// TIA Portal V18 export
// export: Created 2026-06-23T08:49:31.0010641Z, ExportSetting WithDefaults, DisplayName Totally Integrated Automation Portal, DisplayVersion V18, DisplayName TIA Portal Openness, DisplayVersion V18, DisplayName TIA Portal Version Control Interface, DisplayVersion V18, DisplayName STEP 7 Professional, DisplayVersion V18, DisplayName STEP 7 Safety, DisplayVersion V18, DisplayName WinCC Professional, DisplayVersion V18
ORGANIZATION_BLOCK "OB30_PID_PLC1_Bon2"   // OB30, LAD, CyclicInterrupt
{ S7_Optimized_Access := 'TRUE' }
VERSION : 0.1
// stored: AutoNumber true, IsIECCheckEnabled false, SetENOAutomatically false
   VAR_INPUT
      Initial_Call : Bool;   // Initial call of this OB
      Event_Count : Int;   // Events discarded
   END_VAR
BEGIN

REGION Network 1: Initialize PID Bon 2 Kp parameter
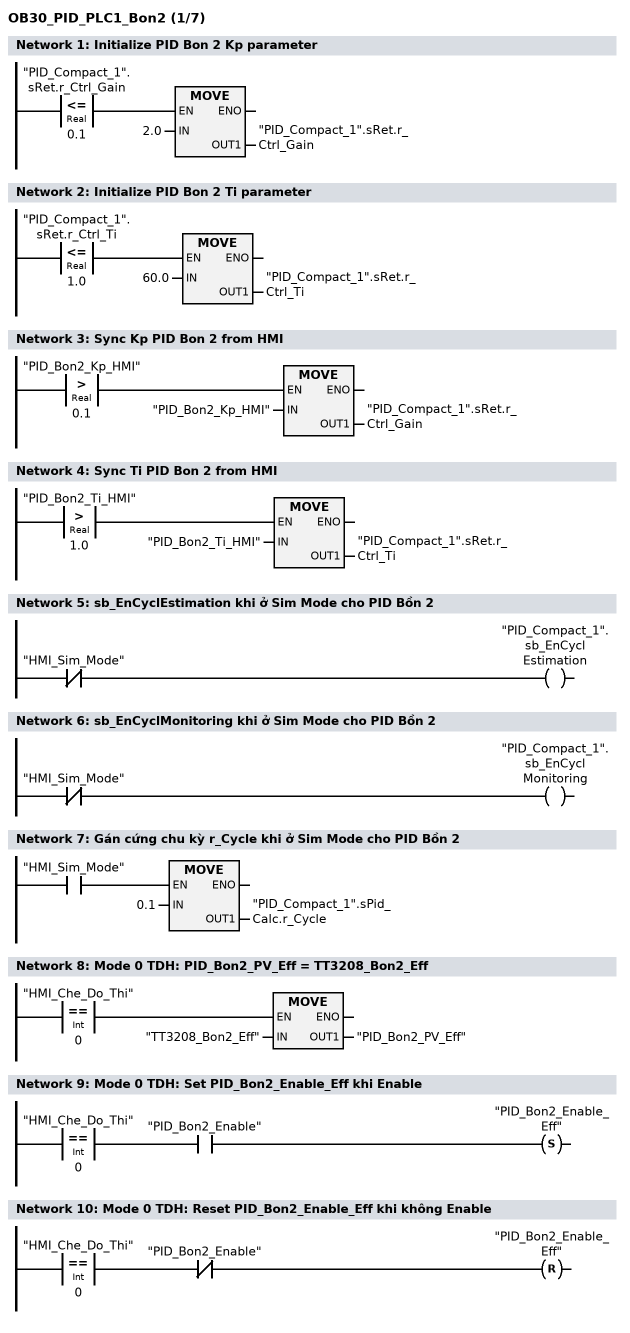
   RUNG wire#powerrail
      { S7_Templates := "SrcType := Real" } LE_Contact(in1 := "PID_Compact_1".sRet.r_Ctrl_Gain, in2 := 0.1)
      { S7_GenerateENO := "TRUE" } Move(in := 2.0, out1 => "PID_Compact_1".sRet.r_Ctrl_Gain)
   END_RUNG
   // the same network as SCL:
   IF "PID_Compact_1".sRet.r_Ctrl_Gain <= 0.1 THEN "PID_Compact_1".sRet.r_Ctrl_Gain := 2.0; END_IF;
END_REGION

REGION Network 2: Initialize PID Bon 2 Ti parameter
   RUNG wire#powerrail
      { S7_Templates := "SrcType := Real" } LE_Contact(in1 := "PID_Compact_1".sRet.r_Ctrl_Ti, in2 := 1.0)
      { S7_GenerateENO := "TRUE" } Move(in := 60.0, out1 => "PID_Compact_1".sRet.r_Ctrl_Ti)
   END_RUNG
   // the same network as SCL:
   IF "PID_Compact_1".sRet.r_Ctrl_Ti <= 1.0 THEN "PID_Compact_1".sRet.r_Ctrl_Ti := 60.0; END_IF;
END_REGION

REGION Network 3: Sync Kp PID Bon 2 from HMI
   RUNG wire#powerrail
      { S7_Templates := "SrcType := Real" } GT_Contact(in1 := "PID_Bon2_Kp_HMI", in2 := 0.1)
      { S7_GenerateENO := "TRUE" } Move(in := "PID_Bon2_Kp_HMI", out1 => "PID_Compact_1".sRet.r_Ctrl_Gain)
   END_RUNG
   // the same network as SCL:
   IF "PID_Bon2_Kp_HMI" > 0.1 THEN "PID_Compact_1".sRet.r_Ctrl_Gain := "PID_Bon2_Kp_HMI"; END_IF;
END_REGION

REGION Network 4: Sync Ti PID Bon 2 from HMI
   RUNG wire#powerrail
      { S7_Templates := "SrcType := Real" } GT_Contact(in1 := "PID_Bon2_Ti_HMI", in2 := 1.0)
      { S7_GenerateENO := "TRUE" } Move(in := "PID_Bon2_Ti_HMI", out1 => "PID_Compact_1".sRet.r_Ctrl_Ti)
   END_RUNG
   // the same network as SCL:
   IF "PID_Bon2_Ti_HMI" > 1.0 THEN "PID_Compact_1".sRet.r_Ctrl_Ti := "PID_Bon2_Ti_HMI"; END_IF;
END_REGION

REGION Network 5: sb_EnCyclEstimation khi ở Sim Mode cho PID Bồn 2
   RUNG wire#powerrail
      I_Contact( "HMI_Sim_Mode" )
      Coil( "PID_Compact_1".sb_EnCyclEstimation )
   END_RUNG
   // the same network as SCL:
   "PID_Compact_1".sb_EnCyclEstimation := NOT "HMI_Sim_Mode";
END_REGION

REGION Network 6: sb_EnCyclMonitoring khi ở Sim Mode cho PID Bồn 2
   RUNG wire#powerrail
      I_Contact( "HMI_Sim_Mode" )
      Coil( "PID_Compact_1".sb_EnCyclMonitoring )
   END_RUNG
   // the same network as SCL:
   "PID_Compact_1".sb_EnCyclMonitoring := NOT "HMI_Sim_Mode";
END_REGION

REGION Network 7: Gán cứng chu kỳ r_Cycle khi ở Sim Mode cho PID Bồn 2
   RUNG wire#powerrail
      Contact( "HMI_Sim_Mode" )
      { S7_GenerateENO := "TRUE" } Move(in := 0.1, out1 => "PID_Compact_1".sPid_Calc.r_Cycle)
   END_RUNG
   // the same network as SCL:
   IF "HMI_Sim_Mode" THEN "PID_Compact_1".sPid_Calc.r_Cycle := 0.1; END_IF;
END_REGION

REGION Network 8: Mode 0 TDH: PID_Bon2_PV_Eff = TT3208_Bon2_Eff
   RUNG wire#powerrail
      { S7_Templates := "SrcType := Int" } EQ_Contact(in1 := "HMI_Che_Do_Thi", in2 := 0)
      { S7_GenerateENO := "TRUE" } Move(in := "TT3208_Bon2_Eff", out1 => "PID_Bon2_PV_Eff")
   END_RUNG
   // the same network as SCL:
   IF "HMI_Che_Do_Thi" = 0 THEN "PID_Bon2_PV_Eff" := "TT3208_Bon2_Eff"; END_IF;
END_REGION

REGION Network 9: Mode 0 TDH: Set PID_Bon2_Enable_Eff khi Enable
   RUNG wire#powerrail
      { S7_Templates := "SrcType := Int" } EQ_Contact(in1 := "HMI_Che_Do_Thi", in2 := 0)
      Contact( "PID_Bon2_Enable" )
      S_Coil( "PID_Bon2_Enable_Eff" )
   END_RUNG
   // the same network as SCL:
   IF ("HMI_Che_Do_Thi" = 0) AND "PID_Bon2_Enable" THEN "PID_Bon2_Enable_Eff" := TRUE; END_IF;
END_REGION

REGION Network 10: Mode 0 TDH: Reset PID_Bon2_Enable_Eff khi không Enable
   RUNG wire#powerrail
      { S7_Templates := "SrcType := Int" } EQ_Contact(in1 := "HMI_Che_Do_Thi", in2 := 0)
      I_Contact( "PID_Bon2_Enable" )
      R_Coil( "PID_Bon2_Enable_Eff" )
   END_RUNG
   // the same network as SCL:
   IF ("HMI_Che_Do_Thi" = 0) AND NOT "PID_Bon2_Enable" THEN "PID_Bon2_Enable_Eff" := FALSE; END_IF;
END_REGION

REGION Network 11: Mode 1 DN: PID_Bon2_PV_Eff = VFD_Bon2_Actual_Speed_Feedback
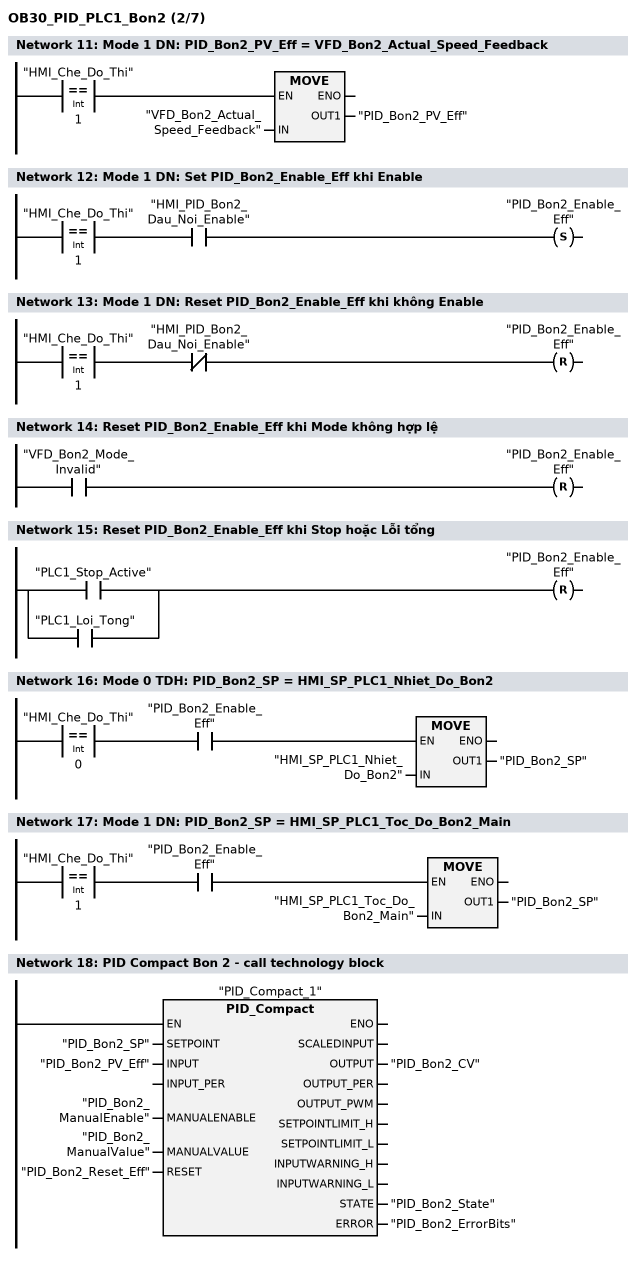
   RUNG wire#powerrail
      { S7_Templates := "SrcType := Int" } EQ_Contact(in1 := "HMI_Che_Do_Thi", in2 := 1)
      { S7_GenerateENO := "TRUE" } Move(in := "VFD_Bon2_Actual_Speed_Feedback", out1 => "PID_Bon2_PV_Eff")
   END_RUNG
   // the same network as SCL:
   IF "HMI_Che_Do_Thi" = 1 THEN "PID_Bon2_PV_Eff" := "VFD_Bon2_Actual_Speed_Feedback"; END_IF;
END_REGION

REGION Network 12: Mode 1 DN: Set PID_Bon2_Enable_Eff khi Enable
   RUNG wire#powerrail
      { S7_Templates := "SrcType := Int" } EQ_Contact(in1 := "HMI_Che_Do_Thi", in2 := 1)
      Contact( "HMI_PID_Bon2_Dau_Noi_Enable" )
      S_Coil( "PID_Bon2_Enable_Eff" )
   END_RUNG
   // the same network as SCL:
   IF ("HMI_Che_Do_Thi" = 1) AND "HMI_PID_Bon2_Dau_Noi_Enable" THEN "PID_Bon2_Enable_Eff" := TRUE; END_IF;
END_REGION

REGION Network 13: Mode 1 DN: Reset PID_Bon2_Enable_Eff khi không Enable
   RUNG wire#powerrail
      { S7_Templates := "SrcType := Int" } EQ_Contact(in1 := "HMI_Che_Do_Thi", in2 := 1)
      I_Contact( "HMI_PID_Bon2_Dau_Noi_Enable" )
      R_Coil( "PID_Bon2_Enable_Eff" )
   END_RUNG
   // the same network as SCL:
   IF ("HMI_Che_Do_Thi" = 1) AND NOT "HMI_PID_Bon2_Dau_Noi_Enable" THEN
       "PID_Bon2_Enable_Eff" := FALSE;
   END_IF;
END_REGION

REGION Network 14: Reset PID_Bon2_Enable_Eff khi Mode không hợp lệ
   RUNG wire#powerrail
      Contact( "VFD_Bon2_Mode_Invalid" )
      R_Coil( "PID_Bon2_Enable_Eff" )
   END_RUNG
   // the same network as SCL:
   IF "VFD_Bon2_Mode_Invalid" THEN "PID_Bon2_Enable_Eff" := FALSE; END_IF;
END_REGION

REGION Network 15: Reset PID_Bon2_Enable_Eff khi Stop hoặc Lỗi tổng
   RUNG wire#powerrail
      Contact( "PLC1_Stop_Active" )
      wire#w1
      R_Coil( "PID_Bon2_Enable_Eff" )
   END_RUNG
   RUNG wire#powerrail
      Contact( "PLC1_Loi_Tong" )
   END_RUNG wire#w1
   // the same network as SCL:
   IF "PLC1_Stop_Active" OR "PLC1_Loi_Tong" THEN "PID_Bon2_Enable_Eff" := FALSE; END_IF;
END_REGION

REGION Network 16: Mode 0 TDH: PID_Bon2_SP = HMI_SP_PLC1_Nhiet_Do_Bon2
   RUNG wire#powerrail
      { S7_Templates := "SrcType := Int" } EQ_Contact(in1 := "HMI_Che_Do_Thi", in2 := 0)
      Contact( "PID_Bon2_Enable_Eff" )
      { S7_GenerateENO := "TRUE" } Move(in := "HMI_SP_PLC1_Nhiet_Do_Bon2", out1 => "PID_Bon2_SP")
   END_RUNG
   // the same network as SCL:
   IF ("HMI_Che_Do_Thi" = 0) AND "PID_Bon2_Enable_Eff" THEN
       "PID_Bon2_SP" := "HMI_SP_PLC1_Nhiet_Do_Bon2";
   END_IF;
END_REGION

REGION Network 17: Mode 1 DN: PID_Bon2_SP = HMI_SP_PLC1_Toc_Do_Bon2_Main
   RUNG wire#powerrail
      { S7_Templates := "SrcType := Int" } EQ_Contact(in1 := "HMI_Che_Do_Thi", in2 := 1)
      Contact( "PID_Bon2_Enable_Eff" )
      { S7_GenerateENO := "TRUE" } Move(in := "HMI_SP_PLC1_Toc_Do_Bon2_Main", out1 => "PID_Bon2_SP")
   END_RUNG
   // the same network as SCL:
   IF ("HMI_Che_Do_Thi" = 1) AND "PID_Bon2_Enable_Eff" THEN
       "PID_Bon2_SP" := "HMI_SP_PLC1_Toc_Do_Bon2_Main";
   END_IF;
END_REGION

REGION Network 18: PID Compact Bon 2 - call technology block
   RUNG wire#powerrail
      "PID_Compact_1".PID_Compact(Setpoint := "PID_Bon2_SP", Input := "PID_Bon2_PV_Eff", Input_PER :=, ManualEnable := "PID_Bon2_ManualEnable", ManualValue := "PID_Bon2_ManualValue", Reset := "PID_Bon2_Reset_Eff", ScaledInput =>, Output => "PID_Bon2_CV", Output_PER =>, Output_PWM =>, SetpointLimit_H =>, SetpointLimit_L =>, InputWarning_H =>, InputWarning_L =>, State => "PID_Bon2_State", Error => "PID_Bon2_ErrorBits")
   END_RUNG
   // the same network as SCL:
   "PID_Compact_1"(Setpoint := "PID_Bon2_SP",   // PID_Compact
                   Input := "PID_Bon2_PV_Eff",
                   ManualEnable := "PID_Bon2_ManualEnable",
                   ManualValue := "PID_Bon2_ManualValue",
                   Reset := "PID_Bon2_Reset_Eff",
                   Output => "PID_Bon2_CV",
                   State => "PID_Bon2_State",
                   Error => "PID_Bon2_ErrorBits");
END_REGION

REGION Network 19: Detect PID Bon 2 Error
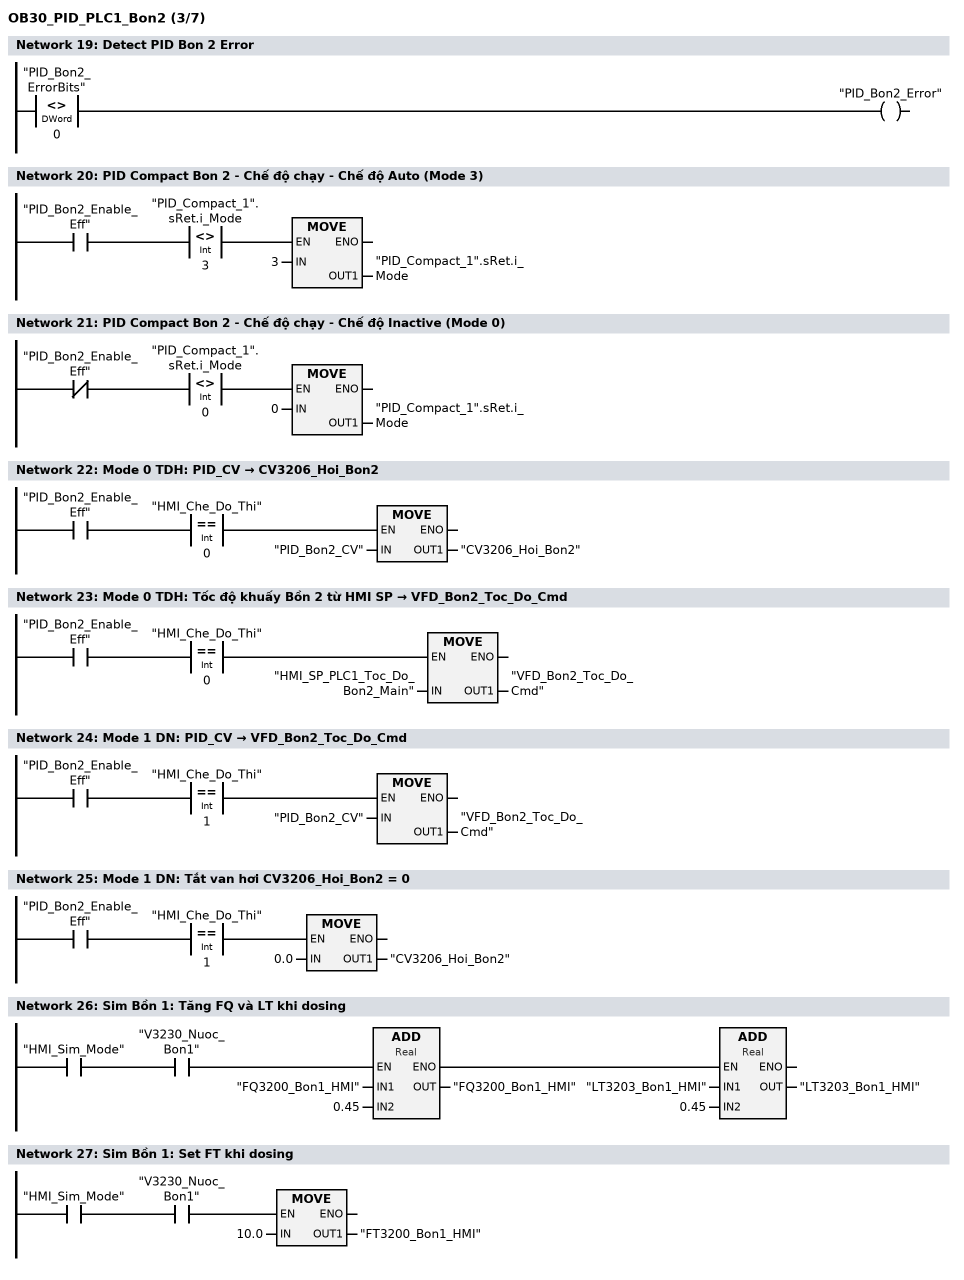
   RUNG wire#powerrail
      { S7_Templates := "SrcType := DWord" } NE_Contact(in1 := "PID_Bon2_ErrorBits", in2 := 0)
      Coil( "PID_Bon2_Error" )
   END_RUNG
   // the same network as SCL:
   "PID_Bon2_Error" := "PID_Bon2_ErrorBits" <> 0;
END_REGION

REGION Network 20: PID Compact Bon 2 - Chế độ chạy - Chế độ Auto (Mode 3)
   RUNG wire#powerrail
      Contact( "PID_Bon2_Enable_Eff" )
      { S7_Templates := "SrcType := Int" } NE_Contact(in1 := "PID_Compact_1".sRet.i_Mode, in2 := 3)
      { S7_GenerateENO := "TRUE" } Move(in := 3, out1 => "PID_Compact_1".sRet.i_Mode)
   END_RUNG
   // the same network as SCL:
   IF "PID_Bon2_Enable_Eff" AND ("PID_Compact_1".sRet.i_Mode <> 3) THEN
       "PID_Compact_1".sRet.i_Mode := 3;
   END_IF;
END_REGION

REGION Network 21: PID Compact Bon 2 - Chế độ chạy - Chế độ Inactive (Mode 0)
   RUNG wire#powerrail
      I_Contact( "PID_Bon2_Enable_Eff" )
      { S7_Templates := "SrcType := Int" } NE_Contact(in1 := "PID_Compact_1".sRet.i_Mode, in2 := 0)
      { S7_GenerateENO := "TRUE" } Move(in := 0, out1 => "PID_Compact_1".sRet.i_Mode)
   END_RUNG
   // the same network as SCL:
   IF NOT "PID_Bon2_Enable_Eff" AND ("PID_Compact_1".sRet.i_Mode <> 0) THEN
       "PID_Compact_1".sRet.i_Mode := 0;
   END_IF;
END_REGION

REGION Network 22: Mode 0 TDH: PID_CV → CV3206_Hoi_Bon2
   RUNG wire#powerrail
      Contact( "PID_Bon2_Enable_Eff" )
      { S7_Templates := "SrcType := Int" } EQ_Contact(in1 := "HMI_Che_Do_Thi", in2 := 0)
      { S7_GenerateENO := "TRUE" } Move(in := "PID_Bon2_CV", out1 => "CV3206_Hoi_Bon2")
   END_RUNG
   // the same network as SCL:
   IF "PID_Bon2_Enable_Eff" AND ("HMI_Che_Do_Thi" = 0) THEN "CV3206_Hoi_Bon2" := "PID_Bon2_CV"; END_IF;
END_REGION

REGION Network 23: Mode 0 TDH: Tốc độ khuấy Bồn 2 từ HMI SP → VFD_Bon2_Toc_Do_Cmd
   RUNG wire#powerrail
      Contact( "PID_Bon2_Enable_Eff" )
      { S7_Templates := "SrcType := Int" } EQ_Contact(in1 := "HMI_Che_Do_Thi", in2 := 0)
      { S7_GenerateENO := "TRUE" } Move(in := "HMI_SP_PLC1_Toc_Do_Bon2_Main", out1 => "VFD_Bon2_Toc_Do_Cmd")
   END_RUNG
   // the same network as SCL:
   IF "PID_Bon2_Enable_Eff" AND ("HMI_Che_Do_Thi" = 0) THEN
       "VFD_Bon2_Toc_Do_Cmd" := "HMI_SP_PLC1_Toc_Do_Bon2_Main";
   END_IF;
END_REGION

REGION Network 24: Mode 1 DN: PID_CV → VFD_Bon2_Toc_Do_Cmd
   RUNG wire#powerrail
      Contact( "PID_Bon2_Enable_Eff" )
      { S7_Templates := "SrcType := Int" } EQ_Contact(in1 := "HMI_Che_Do_Thi", in2 := 1)
      { S7_GenerateENO := "TRUE" } Move(in := "PID_Bon2_CV", out1 => "VFD_Bon2_Toc_Do_Cmd")
   END_RUNG
   // the same network as SCL:
   IF "PID_Bon2_Enable_Eff" AND ("HMI_Che_Do_Thi" = 1) THEN "VFD_Bon2_Toc_Do_Cmd" := "PID_Bon2_CV"; END_IF;
END_REGION

REGION Network 25: Mode 1 DN: Tắt van hơi CV3206_Hoi_Bon2 = 0
   RUNG wire#powerrail
      Contact( "PID_Bon2_Enable_Eff" )
      { S7_Templates := "SrcType := Int" } EQ_Contact(in1 := "HMI_Che_Do_Thi", in2 := 1)
      { S7_GenerateENO := "TRUE" } Move(in := 0.0, out1 => "CV3206_Hoi_Bon2")
   END_RUNG
   // the same network as SCL:
   IF "PID_Bon2_Enable_Eff" AND ("HMI_Che_Do_Thi" = 1) THEN "CV3206_Hoi_Bon2" := 0.0; END_IF;
END_REGION

REGION Network 26: Sim Bồn 1: Tăng FQ và LT khi dosing
   RUNG wire#powerrail
      Contact( "HMI_Sim_Mode" )
      Contact( "V3230_Nuoc_Bon1" )
      { S7_Templates := "SrcType := Real"; S7_GenerateENO := "TRUE" } Add(in1 := "FQ3200_Bon1_HMI", in2 := 0.45, out => "FQ3200_Bon1_HMI")
      { S7_Templates := "SrcType := Real"; S7_GenerateENO := "TRUE" } Add(in1 := "LT3203_Bon1_HMI", in2 := 0.45, out => "LT3203_Bon1_HMI")
   END_RUNG
   // the same network as SCL:
   // ENO of a box is taken as its EN; it also drops when the box reports an error
   IF "HMI_Sim_Mode" AND "V3230_Nuoc_Bon1" THEN
       "FQ3200_Bon1_HMI" := "FQ3200_Bon1_HMI" + 0.45;
       "LT3203_Bon1_HMI" := "LT3203_Bon1_HMI" + 0.45;
   END_IF;
END_REGION

REGION Network 27: Sim Bồn 1: Set FT khi dosing
   RUNG wire#powerrail
      Contact( "HMI_Sim_Mode" )
      Contact( "V3230_Nuoc_Bon1" )
      { S7_GenerateENO := "TRUE" } Move(in := 10.0, out1 => "FT3200_Bon1_HMI")
   END_RUNG
   // the same network as SCL:
   IF "HMI_Sim_Mode" AND "V3230_Nuoc_Bon1" THEN "FT3200_Bon1_HMI" := 10.0; END_IF;
END_REGION

REGION Network 28: Sim Bồn 1: Reset FT khi không dosing
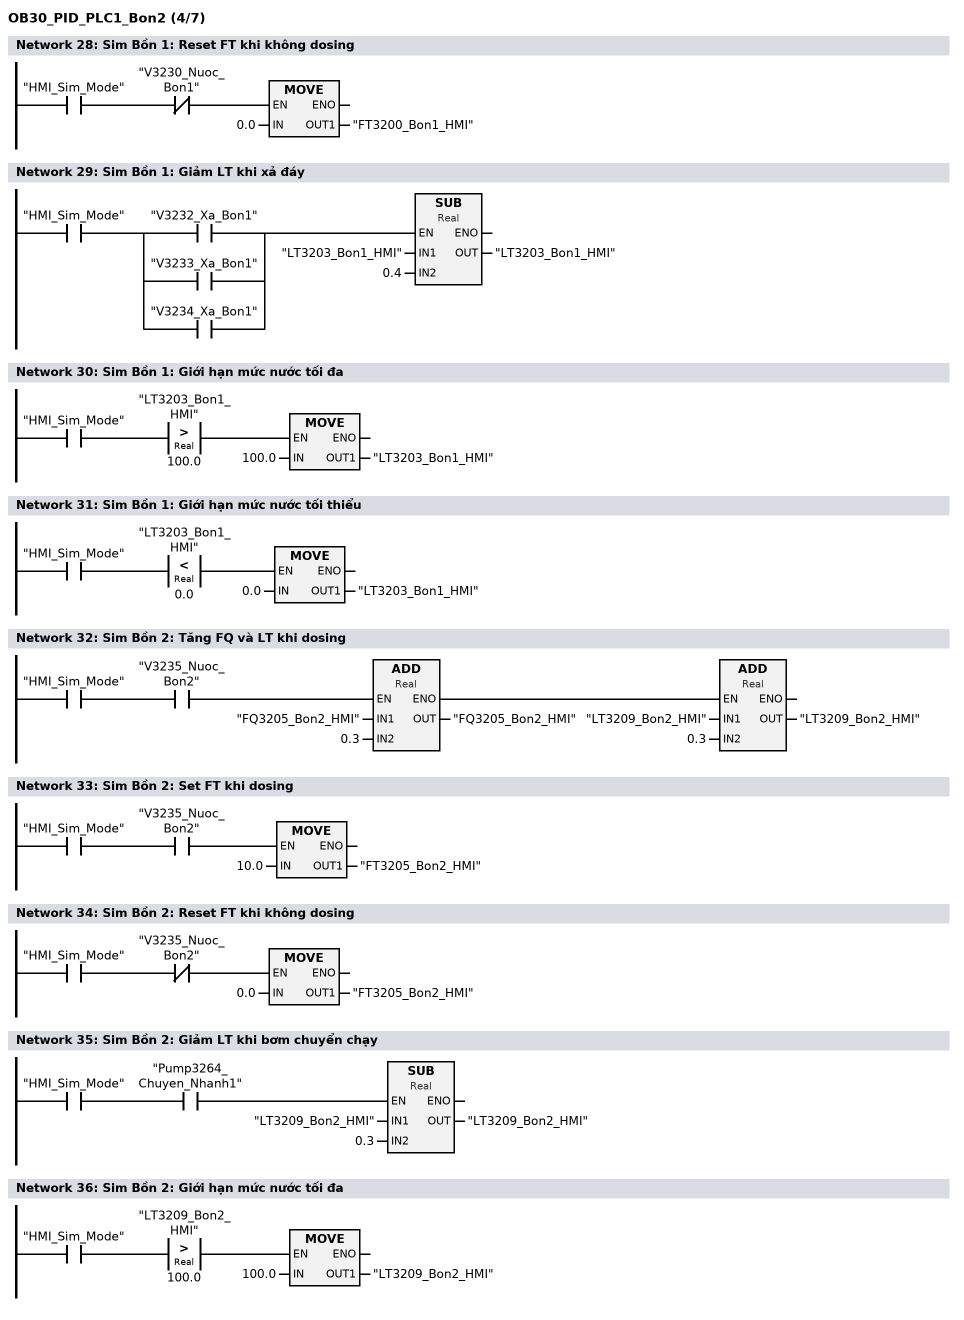
   RUNG wire#powerrail
      Contact( "HMI_Sim_Mode" )
      I_Contact( "V3230_Nuoc_Bon1" )
      { S7_GenerateENO := "TRUE" } Move(in := 0.0, out1 => "FT3200_Bon1_HMI")
   END_RUNG
   // the same network as SCL:
   IF "HMI_Sim_Mode" AND NOT "V3230_Nuoc_Bon1" THEN "FT3200_Bon1_HMI" := 0.0; END_IF;
END_REGION

REGION Network 29: Sim Bồn 1: Giảm LT khi xả đáy
   RUNG wire#powerrail
      Contact( "HMI_Sim_Mode" )
      wire#w1
      Contact( "V3232_Xa_Bon1" )
      wire#w2
      { S7_Templates := "SrcType := Real"; S7_GenerateENO := "TRUE" } Sub(in1 := "LT3203_Bon1_HMI", in2 := 0.4, out => "LT3203_Bon1_HMI")
   END_RUNG
   RUNG wire#w1
      Contact( "V3233_Xa_Bon1" )
   END_RUNG wire#w2
   RUNG wire#w1
      Contact( "V3234_Xa_Bon1" )
   END_RUNG wire#w2
   // the same network as SCL:
   IF "HMI_Sim_Mode" AND ("V3232_Xa_Bon1" OR "V3233_Xa_Bon1" OR "V3234_Xa_Bon1") THEN
       "LT3203_Bon1_HMI" := "LT3203_Bon1_HMI" - 0.4;
   END_IF;
END_REGION

REGION Network 30: Sim Bồn 1: Giới hạn mức nước tối đa
   RUNG wire#powerrail
      Contact( "HMI_Sim_Mode" )
      { S7_Templates := "SrcType := Real" } GT_Contact(in1 := "LT3203_Bon1_HMI", in2 := 100.0)
      { S7_GenerateENO := "TRUE" } Move(in := 100.0, out1 => "LT3203_Bon1_HMI")
   END_RUNG
   // the same network as SCL:
   IF "HMI_Sim_Mode" AND ("LT3203_Bon1_HMI" > 100.0) THEN "LT3203_Bon1_HMI" := 100.0; END_IF;
END_REGION

REGION Network 31: Sim Bồn 1: Giới hạn mức nước tối thiểu
   RUNG wire#powerrail
      Contact( "HMI_Sim_Mode" )
      { S7_Templates := "SrcType := Real" } LT_Contact(in1 := "LT3203_Bon1_HMI", in2 := 0.0)
      { S7_GenerateENO := "TRUE" } Move(in := 0.0, out1 => "LT3203_Bon1_HMI")
   END_RUNG
   // the same network as SCL:
   IF "HMI_Sim_Mode" AND ("LT3203_Bon1_HMI" < 0.0) THEN "LT3203_Bon1_HMI" := 0.0; END_IF;
END_REGION

REGION Network 32: Sim Bồn 2: Tăng FQ và LT khi dosing
   RUNG wire#powerrail
      Contact( "HMI_Sim_Mode" )
      Contact( "V3235_Nuoc_Bon2" )
      { S7_Templates := "SrcType := Real"; S7_GenerateENO := "TRUE" } Add(in1 := "FQ3205_Bon2_HMI", in2 := 0.3, out => "FQ3205_Bon2_HMI")
      { S7_Templates := "SrcType := Real"; S7_GenerateENO := "TRUE" } Add(in1 := "LT3209_Bon2_HMI", in2 := 0.3, out => "LT3209_Bon2_HMI")
   END_RUNG
   // the same network as SCL:
   // ENO of a box is taken as its EN; it also drops when the box reports an error
   IF "HMI_Sim_Mode" AND "V3235_Nuoc_Bon2" THEN
       "FQ3205_Bon2_HMI" := "FQ3205_Bon2_HMI" + 0.3;
       "LT3209_Bon2_HMI" := "LT3209_Bon2_HMI" + 0.3;
   END_IF;
END_REGION

REGION Network 33: Sim Bồn 2: Set FT khi dosing
   RUNG wire#powerrail
      Contact( "HMI_Sim_Mode" )
      Contact( "V3235_Nuoc_Bon2" )
      { S7_GenerateENO := "TRUE" } Move(in := 10.0, out1 => "FT3205_Bon2_HMI")
   END_RUNG
   // the same network as SCL:
   IF "HMI_Sim_Mode" AND "V3235_Nuoc_Bon2" THEN "FT3205_Bon2_HMI" := 10.0; END_IF;
END_REGION

REGION Network 34: Sim Bồn 2: Reset FT khi không dosing
   RUNG wire#powerrail
      Contact( "HMI_Sim_Mode" )
      I_Contact( "V3235_Nuoc_Bon2" )
      { S7_GenerateENO := "TRUE" } Move(in := 0.0, out1 => "FT3205_Bon2_HMI")
   END_RUNG
   // the same network as SCL:
   IF "HMI_Sim_Mode" AND NOT "V3235_Nuoc_Bon2" THEN "FT3205_Bon2_HMI" := 0.0; END_IF;
END_REGION

REGION Network 35: Sim Bồn 2: Giảm LT khi bơm chuyển chạy
   RUNG wire#powerrail
      Contact( "HMI_Sim_Mode" )
      Contact( "Pump3264_Chuyen_Nhanh1" )
      { S7_Templates := "SrcType := Real"; S7_GenerateENO := "TRUE" } Sub(in1 := "LT3209_Bon2_HMI", in2 := 0.3, out => "LT3209_Bon2_HMI")
   END_RUNG
   // the same network as SCL:
   IF "HMI_Sim_Mode" AND "Pump3264_Chuyen_Nhanh1" THEN "LT3209_Bon2_HMI" := "LT3209_Bon2_HMI" - 0.3; END_IF;
END_REGION

REGION Network 36: Sim Bồn 2: Giới hạn mức nước tối đa
   RUNG wire#powerrail
      Contact( "HMI_Sim_Mode" )
      { S7_Templates := "SrcType := Real" } GT_Contact(in1 := "LT3209_Bon2_HMI", in2 := 100.0)
      { S7_GenerateENO := "TRUE" } Move(in := 100.0, out1 => "LT3209_Bon2_HMI")
   END_RUNG
   // the same network as SCL:
   IF "HMI_Sim_Mode" AND ("LT3209_Bon2_HMI" > 100.0) THEN "LT3209_Bon2_HMI" := 100.0; END_IF;
END_REGION

REGION Network 37: Sim Bồn 2: Giới hạn mức nước tối thiểu
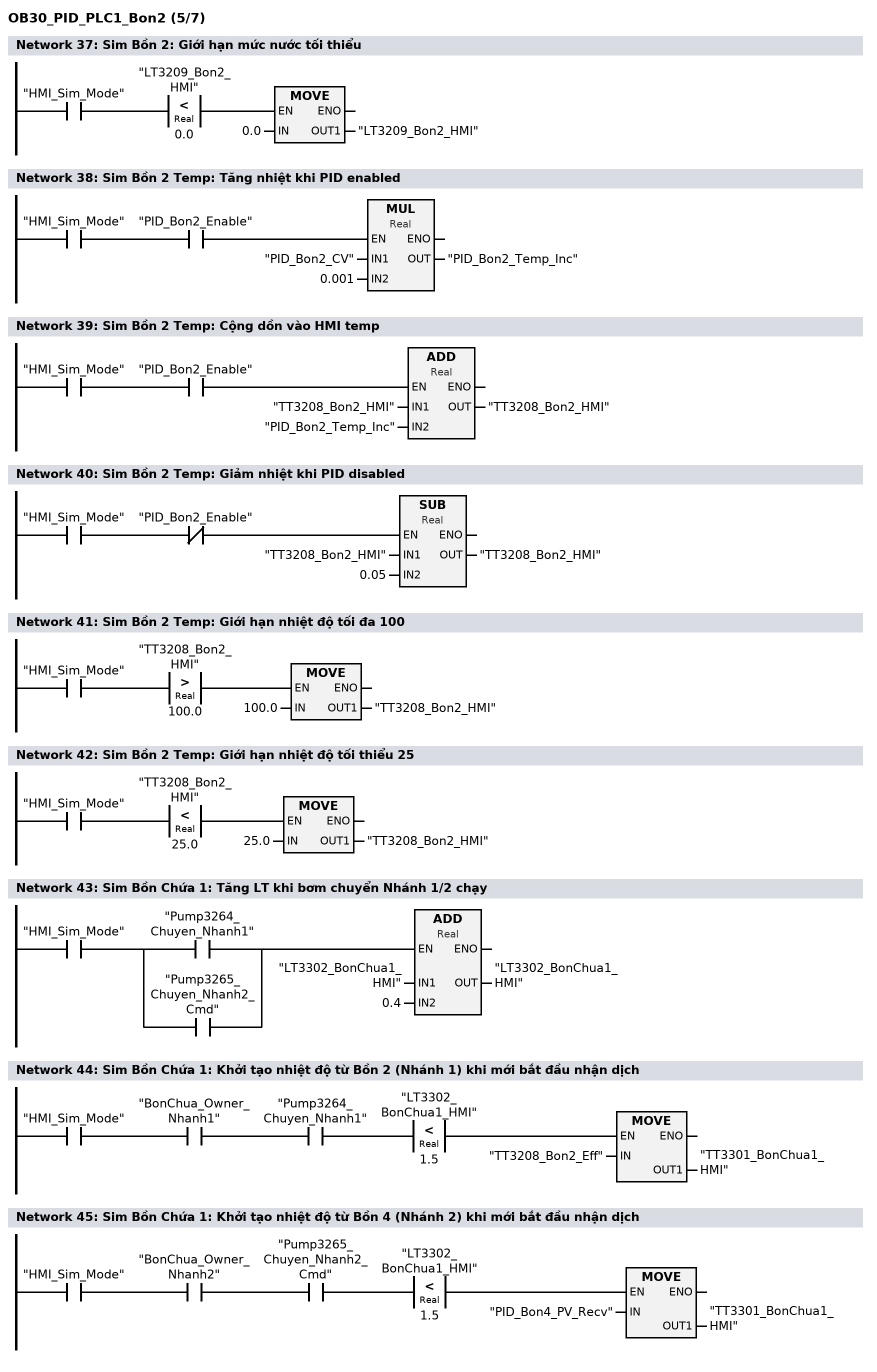
   RUNG wire#powerrail
      Contact( "HMI_Sim_Mode" )
      { S7_Templates := "SrcType := Real" } LT_Contact(in1 := "LT3209_Bon2_HMI", in2 := 0.0)
      { S7_GenerateENO := "TRUE" } Move(in := 0.0, out1 => "LT3209_Bon2_HMI")
   END_RUNG
   // the same network as SCL:
   IF "HMI_Sim_Mode" AND ("LT3209_Bon2_HMI" < 0.0) THEN "LT3209_Bon2_HMI" := 0.0; END_IF;
END_REGION

REGION Network 38: Sim Bồn 2 Temp: Tăng nhiệt khi PID enabled
   RUNG wire#powerrail
      Contact( "HMI_Sim_Mode" )
      Contact( "PID_Bon2_Enable" )
      { S7_Templates := "SrcType := Real"; S7_GenerateENO := "TRUE" } Mul(in1 := "PID_Bon2_CV", in2 := 0.001, out => "PID_Bon2_Temp_Inc")
   END_RUNG
   // the same network as SCL:
   IF "HMI_Sim_Mode" AND "PID_Bon2_Enable" THEN "PID_Bon2_Temp_Inc" := "PID_Bon2_CV" * 0.001; END_IF;
END_REGION

REGION Network 39: Sim Bồn 2 Temp: Cộng dồn vào HMI temp
   RUNG wire#powerrail
      Contact( "HMI_Sim_Mode" )
      Contact( "PID_Bon2_Enable" )
      { S7_Templates := "SrcType := Real"; S7_GenerateENO := "TRUE" } Add(in1 := "TT3208_Bon2_HMI", in2 := "PID_Bon2_Temp_Inc", out => "TT3208_Bon2_HMI")
   END_RUNG
   // the same network as SCL:
   IF "HMI_Sim_Mode" AND "PID_Bon2_Enable" THEN
       "TT3208_Bon2_HMI" := "TT3208_Bon2_HMI" + "PID_Bon2_Temp_Inc";
   END_IF;
END_REGION

REGION Network 40: Sim Bồn 2 Temp: Giảm nhiệt khi PID disabled
   RUNG wire#powerrail
      Contact( "HMI_Sim_Mode" )
      I_Contact( "PID_Bon2_Enable" )
      { S7_Templates := "SrcType := Real"; S7_GenerateENO := "TRUE" } Sub(in1 := "TT3208_Bon2_HMI", in2 := 0.05, out => "TT3208_Bon2_HMI")
   END_RUNG
   // the same network as SCL:
   IF "HMI_Sim_Mode" AND NOT "PID_Bon2_Enable" THEN "TT3208_Bon2_HMI" := "TT3208_Bon2_HMI" - 0.05; END_IF;
END_REGION

REGION Network 41: Sim Bồn 2 Temp: Giới hạn nhiệt độ tối đa 100
   RUNG wire#powerrail
      Contact( "HMI_Sim_Mode" )
      { S7_Templates := "SrcType := Real" } GT_Contact(in1 := "TT3208_Bon2_HMI", in2 := 100.0)
      { S7_GenerateENO := "TRUE" } Move(in := 100.0, out1 => "TT3208_Bon2_HMI")
   END_RUNG
   // the same network as SCL:
   IF "HMI_Sim_Mode" AND ("TT3208_Bon2_HMI" > 100.0) THEN "TT3208_Bon2_HMI" := 100.0; END_IF;
END_REGION

REGION Network 42: Sim Bồn 2 Temp: Giới hạn nhiệt độ tối thiểu 25
   RUNG wire#powerrail
      Contact( "HMI_Sim_Mode" )
      { S7_Templates := "SrcType := Real" } LT_Contact(in1 := "TT3208_Bon2_HMI", in2 := 25.0)
      { S7_GenerateENO := "TRUE" } Move(in := 25.0, out1 => "TT3208_Bon2_HMI")
   END_RUNG
   // the same network as SCL:
   IF "HMI_Sim_Mode" AND ("TT3208_Bon2_HMI" < 25.0) THEN "TT3208_Bon2_HMI" := 25.0; END_IF;
END_REGION

REGION Network 43: Sim Bồn Chứa 1: Tăng LT khi bơm chuyển Nhánh 1/2 chạy
   RUNG wire#powerrail
      Contact( "HMI_Sim_Mode" )
      wire#w1
      Contact( "Pump3264_Chuyen_Nhanh1" )
      wire#w2
      { S7_Templates := "SrcType := Real"; S7_GenerateENO := "TRUE" } Add(in1 := "LT3302_BonChua1_HMI", in2 := 0.4, out => "LT3302_BonChua1_HMI")
   END_RUNG
   RUNG wire#w1
      Contact( "Pump3265_Chuyen_Nhanh2_Cmd" )
   END_RUNG wire#w2
   // the same network as SCL:
   IF "HMI_Sim_Mode" AND ("Pump3264_Chuyen_Nhanh1" OR "Pump3265_Chuyen_Nhanh2_Cmd") THEN
       "LT3302_BonChua1_HMI" := "LT3302_BonChua1_HMI" + 0.4;
   END_IF;
END_REGION

REGION Network 44: Sim Bồn Chứa 1: Khởi tạo nhiệt độ từ Bồn 2 (Nhánh 1) khi mới bắt đầu nhận dịch
   RUNG wire#powerrail
      Contact( "HMI_Sim_Mode" )
      Contact( "BonChua_Owner_Nhanh1" )
      Contact( "Pump3264_Chuyen_Nhanh1" )
      { S7_Templates := "SrcType := Real" } LT_Contact(in1 := "LT3302_BonChua1_HMI", in2 := 1.5)
      { S7_GenerateENO := "TRUE" } Move(in := "TT3208_Bon2_Eff", out1 => "TT3301_BonChua1_HMI")
   END_RUNG
   // the same network as SCL:
   IF "HMI_Sim_Mode" AND "BonChua_Owner_Nhanh1" AND "Pump3264_Chuyen_Nhanh1" AND ("LT3302_BonChua1_HMI" < 1.5) THEN
       "TT3301_BonChua1_HMI" := "TT3208_Bon2_Eff";
   END_IF;
END_REGION

REGION Network 45: Sim Bồn Chứa 1: Khởi tạo nhiệt độ từ Bồn 4 (Nhánh 2) khi mới bắt đầu nhận dịch
   RUNG wire#powerrail
      Contact( "HMI_Sim_Mode" )
      Contact( "BonChua_Owner_Nhanh2" )
      Contact( "Pump3265_Chuyen_Nhanh2_Cmd" )
      { S7_Templates := "SrcType := Real" } LT_Contact(in1 := "LT3302_BonChua1_HMI", in2 := 1.5)
      { S7_GenerateENO := "TRUE" } Move(in := "PID_Bon4_PV_Recv", out1 => "TT3301_BonChua1_HMI")
   END_RUNG
   // the same network as SCL:
   IF "HMI_Sim_Mode" AND "BonChua_Owner_Nhanh2" AND "Pump3265_Chuyen_Nhanh2_Cmd" AND ("LT3302_BonChua1_HMI" < 1.5) THEN
       "TT3301_BonChua1_HMI" := "PID_Bon4_PV_Recv";
   END_IF;
END_REGION

REGION Network 46: Sim Bồn Chứa 1: Giảm nhiệt độ khi bước giải nhiệt active
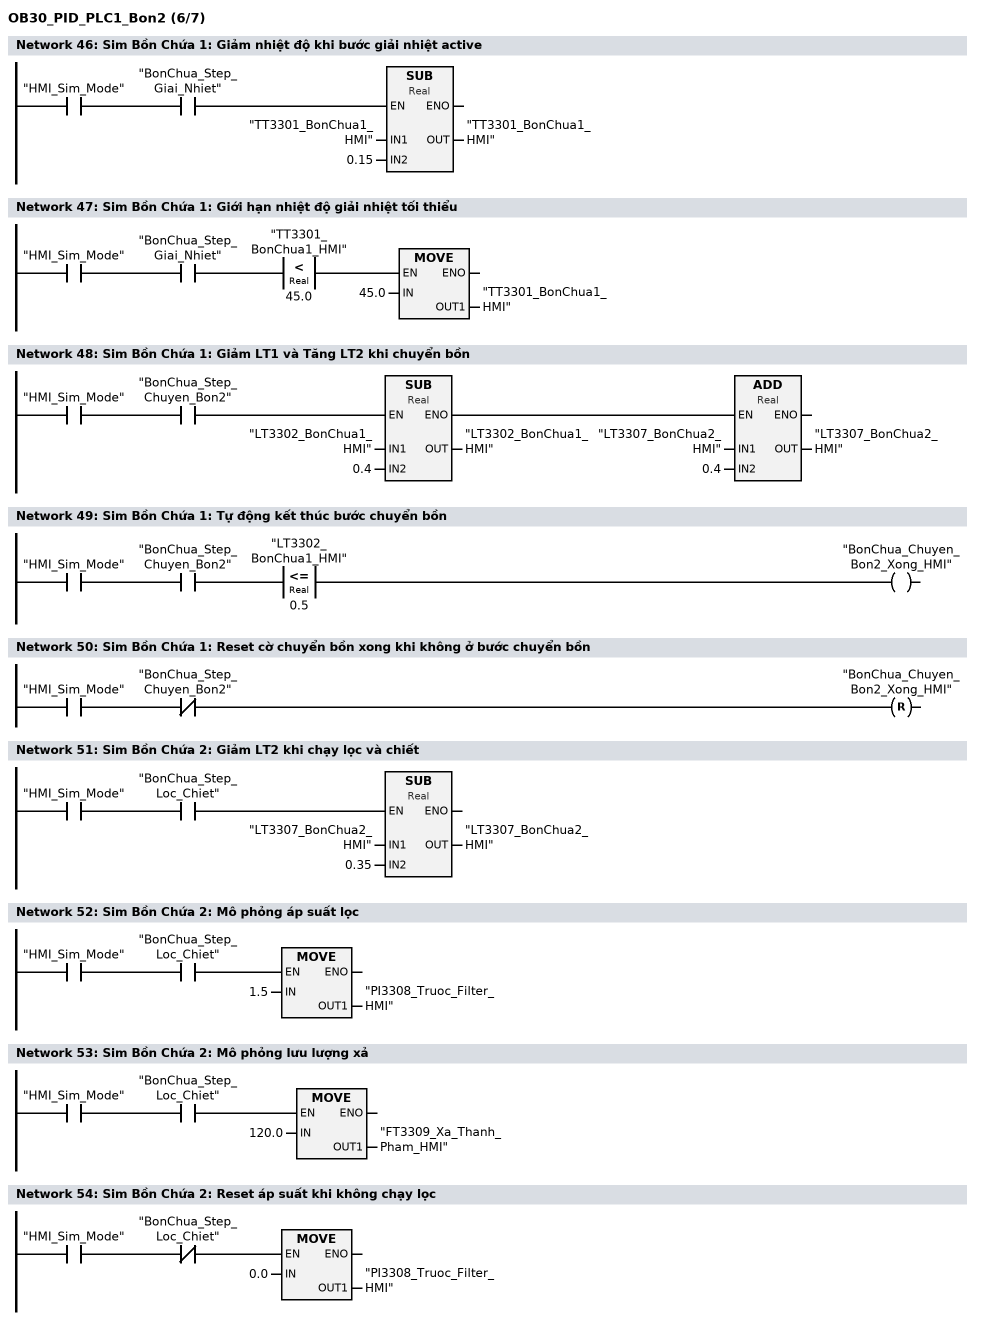
   RUNG wire#powerrail
      Contact( "HMI_Sim_Mode" )
      Contact( "BonChua_Step_Giai_Nhiet" )
      { S7_Templates := "SrcType := Real"; S7_GenerateENO := "TRUE" } Sub(in1 := "TT3301_BonChua1_HMI", in2 := 0.15, out => "TT3301_BonChua1_HMI")
   END_RUNG
   // the same network as SCL:
   IF "HMI_Sim_Mode" AND "BonChua_Step_Giai_Nhiet" THEN
       "TT3301_BonChua1_HMI" := "TT3301_BonChua1_HMI" - 0.15;
   END_IF;
END_REGION

REGION Network 47: Sim Bồn Chứa 1: Giới hạn nhiệt độ giải nhiệt tối thiểu
   RUNG wire#powerrail
      Contact( "HMI_Sim_Mode" )
      Contact( "BonChua_Step_Giai_Nhiet" )
      { S7_Templates := "SrcType := Real" } LT_Contact(in1 := "TT3301_BonChua1_HMI", in2 := 45.0)
      { S7_GenerateENO := "TRUE" } Move(in := 45.0, out1 => "TT3301_BonChua1_HMI")
   END_RUNG
   // the same network as SCL:
   IF "HMI_Sim_Mode" AND "BonChua_Step_Giai_Nhiet" AND ("TT3301_BonChua1_HMI" < 45.0) THEN
       "TT3301_BonChua1_HMI" := 45.0;
   END_IF;
END_REGION

REGION Network 48: Sim Bồn Chứa 1: Giảm LT1 và Tăng LT2 khi chuyển bồn
   RUNG wire#powerrail
      Contact( "HMI_Sim_Mode" )
      Contact( "BonChua_Step_Chuyen_Bon2" )
      { S7_Templates := "SrcType := Real"; S7_GenerateENO := "TRUE" } Sub(in1 := "LT3302_BonChua1_HMI", in2 := 0.4, out => "LT3302_BonChua1_HMI")
      { S7_Templates := "SrcType := Real"; S7_GenerateENO := "TRUE" } Add(in1 := "LT3307_BonChua2_HMI", in2 := 0.4, out => "LT3307_BonChua2_HMI")
   END_RUNG
   // the same network as SCL:
   // ENO of a box is taken as its EN; it also drops when the box reports an error
   IF "HMI_Sim_Mode" AND "BonChua_Step_Chuyen_Bon2" THEN
       "LT3302_BonChua1_HMI" := "LT3302_BonChua1_HMI" - 0.4;
       "LT3307_BonChua2_HMI" := "LT3307_BonChua2_HMI" + 0.4;
   END_IF;
END_REGION

REGION Network 49: Sim Bồn Chứa 1: Tự động kết thúc bước chuyển bồn
   RUNG wire#powerrail
      Contact( "HMI_Sim_Mode" )
      Contact( "BonChua_Step_Chuyen_Bon2" )
      { S7_Templates := "SrcType := Real" } LE_Contact(in1 := "LT3302_BonChua1_HMI", in2 := 0.5)
      Coil( "BonChua_Chuyen_Bon2_Xong_HMI" )
   END_RUNG
   // the same network as SCL:
   "BonChua_Chuyen_Bon2_Xong_HMI" := "HMI_Sim_Mode" AND "BonChua_Step_Chuyen_Bon2" AND ("LT3302_BonChua1_HMI" <= 0.5);
END_REGION

REGION Network 50: Sim Bồn Chứa 1: Reset cờ chuyển bồn xong khi không ở bước chuyển bồn
   RUNG wire#powerrail
      Contact( "HMI_Sim_Mode" )
      I_Contact( "BonChua_Step_Chuyen_Bon2" )
      R_Coil( "BonChua_Chuyen_Bon2_Xong_HMI" )
   END_RUNG
   // the same network as SCL:
   IF "HMI_Sim_Mode" AND NOT "BonChua_Step_Chuyen_Bon2" THEN "BonChua_Chuyen_Bon2_Xong_HMI" := FALSE; END_IF;
END_REGION

REGION Network 51: Sim Bồn Chứa 2: Giảm LT2 khi chạy lọc và chiết
   RUNG wire#powerrail
      Contact( "HMI_Sim_Mode" )
      Contact( "BonChua_Step_Loc_Chiet" )
      { S7_Templates := "SrcType := Real"; S7_GenerateENO := "TRUE" } Sub(in1 := "LT3307_BonChua2_HMI", in2 := 0.35, out => "LT3307_BonChua2_HMI")
   END_RUNG
   // the same network as SCL:
   IF "HMI_Sim_Mode" AND "BonChua_Step_Loc_Chiet" THEN
       "LT3307_BonChua2_HMI" := "LT3307_BonChua2_HMI" - 0.35;
   END_IF;
END_REGION

REGION Network 52: Sim Bồn Chứa 2: Mô phỏng áp suất lọc
   RUNG wire#powerrail
      Contact( "HMI_Sim_Mode" )
      Contact( "BonChua_Step_Loc_Chiet" )
      { S7_GenerateENO := "TRUE" } Move(in := 1.5, out1 => "PI3308_Truoc_Filter_HMI")
   END_RUNG
   // the same network as SCL:
   IF "HMI_Sim_Mode" AND "BonChua_Step_Loc_Chiet" THEN "PI3308_Truoc_Filter_HMI" := 1.5; END_IF;
END_REGION

REGION Network 53: Sim Bồn Chứa 2: Mô phỏng lưu lượng xả
   RUNG wire#powerrail
      Contact( "HMI_Sim_Mode" )
      Contact( "BonChua_Step_Loc_Chiet" )
      { S7_GenerateENO := "TRUE" } Move(in := 120.0, out1 => "FT3309_Xa_Thanh_Pham_HMI")
   END_RUNG
   // the same network as SCL:
   IF "HMI_Sim_Mode" AND "BonChua_Step_Loc_Chiet" THEN "FT3309_Xa_Thanh_Pham_HMI" := 120.0; END_IF;
END_REGION

REGION Network 54: Sim Bồn Chứa 2: Reset áp suất khi không chạy lọc
   RUNG wire#powerrail
      Contact( "HMI_Sim_Mode" )
      I_Contact( "BonChua_Step_Loc_Chiet" )
      { S7_GenerateENO := "TRUE" } Move(in := 0.0, out1 => "PI3308_Truoc_Filter_HMI")
   END_RUNG
   // the same network as SCL:
   IF "HMI_Sim_Mode" AND NOT "BonChua_Step_Loc_Chiet" THEN "PI3308_Truoc_Filter_HMI" := 0.0; END_IF;
END_REGION

REGION Network 55: Sim Bồn Chứa 2: Reset lưu lượng xả khi không chạy lọc
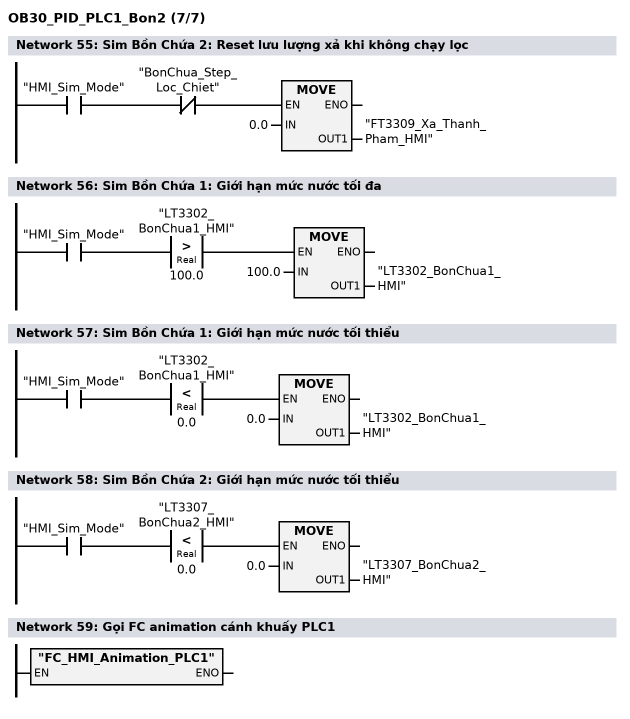
   RUNG wire#powerrail
      Contact( "HMI_Sim_Mode" )
      I_Contact( "BonChua_Step_Loc_Chiet" )
      { S7_GenerateENO := "TRUE" } Move(in := 0.0, out1 => "FT3309_Xa_Thanh_Pham_HMI")
   END_RUNG
   // the same network as SCL:
   IF "HMI_Sim_Mode" AND NOT "BonChua_Step_Loc_Chiet" THEN "FT3309_Xa_Thanh_Pham_HMI" := 0.0; END_IF;
END_REGION

REGION Network 56: Sim Bồn Chứa 1: Giới hạn mức nước tối đa
   RUNG wire#powerrail
      Contact( "HMI_Sim_Mode" )
      { S7_Templates := "SrcType := Real" } GT_Contact(in1 := "LT3302_BonChua1_HMI", in2 := 100.0)
      { S7_GenerateENO := "TRUE" } Move(in := 100.0, out1 => "LT3302_BonChua1_HMI")
   END_RUNG
   // the same network as SCL:
   IF "HMI_Sim_Mode" AND ("LT3302_BonChua1_HMI" > 100.0) THEN "LT3302_BonChua1_HMI" := 100.0; END_IF;
END_REGION

REGION Network 57: Sim Bồn Chứa 1: Giới hạn mức nước tối thiểu
   RUNG wire#powerrail
      Contact( "HMI_Sim_Mode" )
      { S7_Templates := "SrcType := Real" } LT_Contact(in1 := "LT3302_BonChua1_HMI", in2 := 0.0)
      { S7_GenerateENO := "TRUE" } Move(in := 0.0, out1 => "LT3302_BonChua1_HMI")
   END_RUNG
   // the same network as SCL:
   IF "HMI_Sim_Mode" AND ("LT3302_BonChua1_HMI" < 0.0) THEN "LT3302_BonChua1_HMI" := 0.0; END_IF;
END_REGION

REGION Network 58: Sim Bồn Chứa 2: Giới hạn mức nước tối thiểu
   RUNG wire#powerrail
      Contact( "HMI_Sim_Mode" )
      { S7_Templates := "SrcType := Real" } LT_Contact(in1 := "LT3307_BonChua2_HMI", in2 := 0.0)
      { S7_GenerateENO := "TRUE" } Move(in := 0.0, out1 => "LT3307_BonChua2_HMI")
   END_RUNG
   // the same network as SCL:
   IF "HMI_Sim_Mode" AND ("LT3307_BonChua2_HMI" < 0.0) THEN "LT3307_BonChua2_HMI" := 0.0; END_IF;
END_REGION

REGION Network 59: Gọi FC animation cánh khuấy PLC1
   RUNG wire#powerrail
      "FC_HMI_Animation_PLC1"()
   END_RUNG
   // the same network as SCL:
   "FC_HMI_Animation_PLC1"();
END_REGION
END_ORGANIZATION_BLOCK
